//-----------------------------------------------------------------------------------------
//
//                  				ST_Message
//
//								Variables message			
//-----------------------------------------------------------------------------------------
//
//Auteur: G.GOETZ (inspired by S.MANTZER)
//Création: 21.01.2026
//Dernière modification : 21.01.2026 (G.GOETZ)
//       			
//-----------------------------------------------------------------------------------------
//
//     							Liste des modifications  	
//
// 21.01.2026 (G.GOETZ) -> Création		
//-----------------------------------------------------------------------------------------

TYPE ST_Message :
STRUCT
		
	(** FB **)
	fbMessage : FB_TcMessage;

END_STRUCT
END_TYPE

(* stored: Version 1.1.0.1, ProductVersion 3.1.4024.13
   DUT ST_Message: Id {aae68cd3-57d7-46f2-b7f9-6579667ee5c0} *)
